{attribute 'no-analysis'}
TYPE ST_EL3443_VariantValues :
STRUCT
	astLx 			: ARRAY[1..3] OF ST_EL3443_VariantLx;
	stTotal 		: ST_EL3443_VariantTotal;
END_STRUCT
END_TYPE

(* stored: Version 1.1.0.1, ProductVersion 3.1.4024.4
   DUT ST_EL3443_VariantValues: Id {6b275d55-c1cc-4fab-9374-872387b1ece1} *)
